// TIA Portal V20 export
DATA_BLOCK "LBP_InternalDB1020"   // DB1020
TITLE = Internal DB for basic program / DB interne pour programme de base
// DB only for internal use in the basic program / DB réservé à l'utilisation interne dans le programme de base
// stored: AutoNumber false, InstanceOfName LBP_InternalFB1020, InstanceOfType FB
"LBP_InternalFB1020"
   // VAR_INPUT
   //    IN1 : UDInt;
   //    IN2 : UDInt;
   //    IN3 : Word;
   //    IN4 : Variant;
   //    IN5 : Variant;
   //    IN6 : Variant;
   //    IN7 : Variant;
   //    IN8 : Variant;
   //    IN9 : Variant;
   //    IN10 : Variant;
   //    IN11 : Variant;
   //    IN12 : Variant;
   // END_VAR
   // VAR_OUTPUT
   //    OUT1 : Bool;
   //    OUT2 : DWord;
   //    OUT3 : UInt;
   // END_VAR
   // VAR
   //    LBP_AlarmType_ErrMsg { S7_SetPoint := 'True'} : Diag_Alarm;
   //    LBP_AlarmType_OpMsg { S7_SetPoint := 'True'} : Diag_Alarm;
   //    LBP_AlarmType_InfoMsg { S7_SetPoint := 'True'} : Diag_Alarm;
   //    LBP_DB2AlarmType_ErrMsg { S7_SetPoint := 'True'} : Diag_Alarm;
   //    LBP_DB2AlarmType_OpMsg { S7_SetPoint := 'True'} : Diag_Alarm;
   //    LBP_DB2AlarmType_InfoMsg { S7_SetPoint := 'True'} : Diag_Alarm;
   //    LBP_UserAlarmType_ErrMsg { S7_SetPoint := 'True'} : Diag_Alarm;
   //    LBP_UserAlarmType_OpMsg { S7_SetPoint := 'True'} : Diag_Alarm;
   //    LBP_UserAlarmType_InfoMsg { S7_SetPoint := 'True'} : Diag_Alarm;
   //    LBP_UserAlarmType_AckMsg { S7_SetPoint := 'True'} : Diag_Alarm;
   //    s_strct_DB2AddressLastCycle : Struct
   //       LwByteAddress : DInt;
   //       LwBitAddress : DInt;
   //    END_STRUCT;
   //    s_DB2_MaxScanByteUser : DInt;
   //    s_DB7_Params : Struct
   //       MaxAxis : Int;
   //       MaxChan : Int;
   //       MsgUser : Int;
   //       ExtendChanAxMsg : Bool;
   //       ActivChan : Array[1..10] of Bool;
   //       ActivAxis : Array[1..31] of Bool;
   //    END_STRUCT;
   //    s_firstScanFinished : Bool;
   //    s_FC10_Quit : Struct
   //       QuitEdge : Bool;
   //       LwByteAddress : DInt;
   //       DB2ScanFinished : Bool;
   //    END_STRUCT;
   //    s_CounterActiveDB2Alarms : UInt;
   //    s_FC10_ToUserIf_OLD : Bool;
   // END_VAR
BEGIN
END_DATA_BLOCK
